# EPICS substitutions: evrMrmApp/Db/evr-cpci-230.substitutions
# Record set for a EVR-cPCI-230
#
# Macros:
#  DEVICE = Event receiver / timing card name (same as mrmEvrSetupVME()) Eg. EVR0
#  SYS = System name (ie SR-TM)
#
# Record names have the general forms:
#  $(SYS)-$(DEVICE):Signal-SD

file "evr-base.template"
{pattern
{ SYS,      DEVICE,     EVNT1HZ}
{"$(SYS)", "$(DEVICE)", 125}
}

file "sfp.template"
{
{SYS="$(SYS)", DEVICE="$(DEVICE)", ID="0"}
}

file "flash.template"
{
{SYS="$(SYS)", DEVICE="$(DEVICE)"}
}

file "evr-prescaler.template"
{pattern
{ SYS,      DEVICE,     ID, MAX}
{"$(SYS)", "$(DEVICE)", 0, "0xffffffff"}
{"$(SYS)", "$(DEVICE)", 1, "0xffffffff"}
{"$(SYS)", "$(DEVICE)", 2, "0xffffffff"}
}

# Pulse generators w/o a prescaler set NOPS=1
file "evr-pulser.template"
{pattern
{ SYS,      DEVICE,     ID,  DMAX,       WMAX,          PMAX,    NOPS}
{"$(SYS)", "$(DEVICE)", 0,  "0xffffffff", "0xffffffff", "0xffff", 0}
{"$(SYS)", "$(DEVICE)", 1,  "0xffffffff", "0xffffffff", "0xffff", 0}
{"$(SYS)", "$(DEVICE)", 2,  "0xffffffff", "0xffffffff", "0xffff", 0}
{"$(SYS)", "$(DEVICE)", 3,  "0xffffffff", "0xffffffff", "0xffff", 0}
{"$(SYS)", "$(DEVICE)", 4,  "0xffffffff", "0xffff",     "1",      1}
{"$(SYS)", "$(DEVICE)", 5,  "0xffffffff", "0xffff",     "1",      1}
{"$(SYS)", "$(DEVICE)", 6,  "0xffffffff", "0xffff",     "1",      1}
{"$(SYS)", "$(DEVICE)", 7,  "0xffffffff", "0xffff",     "1",      1}
{"$(SYS)", "$(DEVICE)", 8,  "0xffffffff", "0xffff",     "1",      1}
{"$(SYS)", "$(DEVICE)", 9,  "0xffffffff", "0xffff",     "1",      1}
}

file "evr-in.template"
{pattern
{ SYS,      DEVICE,     ID,  DESC}
{"$(SYS)", "$(DEVICE)", 0,  "IN0 (TTL)"}
{"$(SYS)", "$(DEVICE)", 1,  "IN1 (TTL)"}
}

file "evr-out.template"
{pattern
{ SYS,      DEVICE,      OBJ,    		 	ID,   DESC}
{"$(SYS)", "$(DEVICE)", "FrontUnivOut", 	0,   "UNIV0"}
{"$(SYS)", "$(DEVICE)", "FrontUnivOut", 	1,   "UNIV1"}
{"$(SYS)", "$(DEVICE)", "FrontUnivOut", 	2,   "UNIV2"}
{"$(SYS)", "$(DEVICE)", "FrontUnivOut", 	3,   "UNIV3"}
}
